// TIA Portal V18 export
// export: Created 2026-06-12T02:00:00Z, ExportSetting WithDefaults, DisplayName Totally Integrated Automation Portal, DisplayVersion V18, DisplayName TIA Portal Openness, DisplayVersion V18
TagTable "AI_B7_Tags"
  AI_B7_K03_PT02_Pressure : Real  (PLC tag AI_B7_K03_PT02_Pressure, HMI_Connection_1, 1 s)   // PRESSURE 7-8 bar
  AI_B7_K03_TT04_Temp : Real  (PLC tag AI_B7_K03_TT04_Temp, HMI_Connection_1, 1 s)   // TEMP 50-80 °C
  AI_B7_K03_TT05_Temp : Real  (PLC tag AI_B7_K03_TT05_Temp, HMI_Connection_1, 1 s)   // TEMP 50-80 °C
  AI_B7_K03_TT06_Temp : Real  (PLC tag AI_B7_K03_TT06_Temp, HMI_Connection_1, 1 s)   // TEMP 50-80 °C
  AI_B7_K03_TT07_Temp : Real  (PLC tag AI_B7_K03_TT07_Temp, HMI_Connection_1, 1 s)   // TEMP 50-80 °C
  AI_B7_K03_PT07_Pressure : Real  (PLC tag AI_B7_K03_PT07_Pressure, HMI_Connection_1, 1 s)   // PRESSURE 7-8 bar
  AI_B7_K03_FT03_Flow : Real  (PLC tag AI_B7_K03_FT03_Flow, HMI_Connection_1, 1 s)   // FLOW 100-200 L/h
  AI_B7_K03_Density_1 : Real  (PLC tag AI_B7_K03_Density_1, HMI_Connection_1, 1 s)   // COUNT 800-1000 kg/m3
  AI_B7_K03_LT01_Level : Real  (PLC tag AI_B7_K03_LT01_Level, HMI_Connection_1, 1 s)   // LEVEL 20-80 cm
  AI_B7_K03_LT02_Level : Real  (PLC tag AI_B7_K03_LT02_Level, HMI_Connection_1, 1 s)   // LEVEL 20-80 cm
  AI_B7_K03_TT01_Temp : Real  (PLC tag AI_B7_K03_TT01_Temp, HMI_Connection_1, 1 s)   // TEMP 50-80 °C
  AI_B7_K03_TT02_Temp : Real  (PLC tag AI_B7_K03_TT02_Temp, HMI_Connection_1, 1 s)   // TEMP 50-80 °C
  AI_B7_Reboiler_PV : Real  (PLC tag AI_B7_Reboiler_PV, HMI_Connection_1, 1 s)   // FLOW 100-200 L/h
  AI_B7_Reboiler_SP : Real  (PLC tag AI_B7_Reboiler_SP, HMI_Connection_1, 1 s)   // FLOW 100-200 L/h
  AI_B7_Reboiler_CV : Real  (PLC tag AI_B7_Reboiler_CV, HMI_Connection_1, 1 s)   // PERCENT 20-80 %
  AI_B7_HE03_Primary_Temp : Real  (PLC tag AI_B7_HE03_Primary_Temp, HMI_Connection_1, 1 s)   // TEMP 50-80 °C
  AI_B7_HE03_Secondary_Temp : Real  (PLC tag AI_B7_HE03_Secondary_Temp, HMI_Connection_1, 1 s)   // TEMP 50-80 °C
  AI_B7_K03_L08_Level : Real  (PLC tag AI_B7_K03_L08_Level, HMI_Connection_1, 1 s)   // LEVEL 20-80 cm
  AI_B7_K03_L06_Level : Real  (PLC tag AI_B7_K03_L06_Level, HMI_Connection_1, 1 s)   // LEVEL 20-80 cm
  AI_B7_K03_L05_Level : Real  (PLC tag AI_B7_K03_L05_Level, HMI_Connection_1, 1 s)   // LEVEL 20-80 cm
  AI_B7_K03_L07_Level : Real  (PLC tag AI_B7_K03_L07_Level, HMI_Connection_1, 1 s)   // LEVEL 20-80 cm
  AI_B7_K03_L04_Level : Real  (PLC tag AI_B7_K03_L04_Level, HMI_Connection_1, 1 s)   // LEVEL 20-80 cm
  AI_B7_K03_L03_Level : Real  (PLC tag AI_B7_K03_L03_Level, HMI_Connection_1, 1 s)   // LEVEL 20-80 cm
  AI_B7_V03A_Density : Real  (PLC tag AI_B7_V03A_Density, HMI_Connection_1, 1 s)   // COUNT 800-1000 kg/m3
  AI_B7_Kettle_Flow_SP : Real  (PLC tag AI_B7_Kettle_Flow_SP, HMI_Connection_1, 1 s)   // FLOW 100-200 kg/h
  AI_B7_Keboiler_Flow_SP : Real  (PLC tag AI_B7_Keboiler_Flow_SP, HMI_Connection_1, 1 s)   // FLOW 100-200 kg/h
  AI_B7_Reflux_Time_SP : Real  (PLC tag AI_B7_Reflux_Time_SP, HMI_Connection_1, 1 s)   // COUNT 0-60 Min
  AI_B7_Time_Remain : Real  (PLC tag AI_B7_Time_Remain, HMI_Connection_1, 1 s)   // COUNT 0-60 Min
  AI_B7_RD_Level_SP : Real  (PLC tag AI_B7_RD_Level_SP, HMI_Connection_1, 1 s)   // LEVEL 20-80 cm
  AI_B7_Reflux_Flow_SP : Real  (PLC tag AI_B7_Reflux_Flow_SP, HMI_Connection_1, 1 s)   // FLOW 100-200 L/h
  AI_B7_Collection_SP : Real  (PLC tag AI_B7_Collection_SP, HMI_Connection_1, 1 s)   // FLOW 100-200 L/h
  AI_B7_Total_Flowrate : Real  (PLC tag AI_B7_Total_Flowrate, HMI_Connection_1, 1 s)   // FLOW 100-200 L/h
  AI_B7_ML_Qty_SP : Real  (PLC tag AI_B7_ML_Qty_SP, HMI_Connection_1, 1 s)   // COUNT 0-600 L
  AI_B7_ML_Qty_Total : Real  (PLC tag AI_B7_ML_Qty_Total, HMI_Connection_1, 1 s)   // COUNT 0-600 L
  AI_B7_Material_Code : Real  (PLC tag AI_B7_Material_Code, HMI_Connection_1, 1 s)   // COUNT 0-99
  AI_B7_Stage_Number : Real  (PLC tag AI_B7_Stage_Number, HMI_Connection_1, 1 s)   // COUNT 0-20
  AI_B7_Batch_Number : Real  (PLC tag AI_B7_Batch_Number, HMI_Connection_1, 1 s)   // COUNT 0-9999
  AI_B7_Current_User_ID : Real  (PLC tag AI_B7_Current_User_ID, HMI_Connection_1, 1 s)   // COUNT 0-999
  AI_B7_K_05_L_704_HI : Real  (PLC tag AI_B7_K_05_L_704_HI, HMI_Connection_1, 1 s)   // LEVEL 20-80 cm
  AI_B7_Density_SP : Real  (PLC tag AI_B7_Density_SP, HMI_Connection_1, 1 s)   // COUNT 800-1000 kg/m3
  AI_B7_CTS_Flow_1 : Real  (PLC tag AI_B7_CTS_Flow_1, HMI_Connection_1, 1 s)   // FLOW 100-200 kg/h
  AI_B7_CTS_Flow_2 : Real  (PLC tag AI_B7_CTS_Flow_2, HMI_Connection_1, 1 s)   // FLOW 100-200 kg/h
  AI_B7_Steam_PT01_Temp : Real  (PLC tag AI_B7_Steam_PT01_Temp, HMI_Connection_1, 1 s)   // TEMP 50-80 °C
  AI_B7_Steam_PT02_Temp : Real  (PLC tag AI_B7_Steam_PT02_Temp, HMI_Connection_1, 1 s)   // TEMP 50-80 °C
  AI_B7_CWS_TT01_Temp : Real  (PLC tag AI_B7_CWS_TT01_Temp, HMI_Connection_1, 1 s)   // TEMP 50-80 °C
  AI_B7_CWS_TT02_Temp : Real  (PLC tag AI_B7_CWS_TT02_Temp, HMI_Connection_1, 1 s)   // TEMP 50-80 °C
  AI_B7_CWS_TT03_Temp : Real  (PLC tag AI_B7_CWS_TT03_Temp, HMI_Connection_1, 1 s)   // TEMP 50-80 °C
  AI_B7_CWAR_TT01_Temp : Real  (PLC tag AI_B7_CWAR_TT01_Temp, HMI_Connection_1, 1 s)   // TEMP 50-80 °C
  AI_B7_CWAR_TT02_Temp : Real  (PLC tag AI_B7_CWAR_TT02_Temp, HMI_Connection_1, 1 s)   // TEMP 50-80 °C
  AI_B7_CWAR_TT03_Temp : Real  (PLC tag AI_B7_CWAR_TT03_Temp, HMI_Connection_1, 1 s)   // TEMP 50-80 °C
  AI_B7_CWAR_TT04_Temp : Real  (PLC tag AI_B7_CWAR_TT04_Temp, HMI_Connection_1, 1 s)   // TEMP 50-80 °C
  AI_B7_K03_CV01_PV : Real  (PLC tag AI_B7_K03_CV01_PV, HMI_Connection_1, 1 s)   // PERCENT 20-80 %
  AI_B7_K03_CV01_SP : Real  (PLC tag AI_B7_K03_CV01_SP, HMI_Connection_1, 1 s)   // PERCENT 20-80 %
  AI_B7_K03_CV01_CV : Real  (PLC tag AI_B7_K03_CV01_CV, HMI_Connection_1, 1 s)   // PERCENT 20-80 %
  AI_B7_Steam_CV01_PV : Real  (PLC tag AI_B7_Steam_CV01_PV, HMI_Connection_1, 1 s)   // PERCENT 20-80 %
  AI_B7_Steam_CV01_SP : Real  (PLC tag AI_B7_Steam_CV01_SP, HMI_Connection_1, 1 s)   // PERCENT 20-80 %
  AI_B7_Steam_CV01_CV : Real  (PLC tag AI_B7_Steam_CV01_CV, HMI_Connection_1, 1 s)   // PERCENT 20-80 %
  AI_B7_K03_Jacket_PV : Real  (PLC tag AI_B7_K03_Jacket_PV, HMI_Connection_1, 1 s)   // TEMP 50-80 °C
  AI_B7_K03_Jacket_SP : Real  (PLC tag AI_B7_K03_Jacket_SP, HMI_Connection_1, 1 s)   // TEMP 50-80 °C
  AI_B7_K03_Jacket_CV : Real  (PLC tag AI_B7_K03_Jacket_CV, HMI_Connection_1, 1 s)   // PERCENT 20-80 %
  AI_B7_CHWR_TT01_Temp : Real  (PLC tag AI_B7_CHWR_TT01_Temp, HMI_Connection_1, 1 s)   // TEMP 50-80 °C
  AI_B7_CHWR_TT02_Temp : Real  (PLC tag AI_B7_CHWR_TT02_Temp, HMI_Connection_1, 1 s)   // TEMP 50-80 °C
  AI_B7_CHWS_TT01_Temp : Real  (PLC tag AI_B7_CHWS_TT01_Temp, HMI_Connection_1, 1 s)   // TEMP 50-80 °C
  AI_B7_CHWS_TT02_Temp : Real  (PLC tag AI_B7_CHWS_TT02_Temp, HMI_Connection_1, 1 s)   // TEMP 50-80 °C
  AI_B7_K03_TT03_Temp : Real  (PLC tag AI_B7_K03_TT03_Temp, HMI_Connection_1, 1 s)   // TEMP 50-80 °C
